// Mitsubishi GX Works2 project: DanNhanFX3G   PLC: FX3G

// global labels: Global1
VAR_GLOBAL
  SIGNAL_BOTTLE AT X000 : BOOL;
  SIGNAL_LABEL AT X001 : BOOL;
  EMERG AT X007 : BOOL;
  LABEL_PLS AT Y000 : BOOL;
  LABEL_DIR AT Y003 : BOOL;
  PushManLabel_F AT M200 : BOOL;
  PushManLabel_R AT M201 : BOOL;
  ModeAuto AT M206 : BOOL;
  Alarm AT M207 : BOOL;
  Operation AT M208 : BOOL;
  Speed_Label AT D200 : REAL;
  Length_Label AT D202 : REAL;
  Reset AT M209 : BOOL;
  Restore AT M210 : BOOL;
  LABEL_ENB AT Y004 : BOOL;
  GIRD_PLS AT Y001 : BOOL;
  RULO_PLS AT Y002 : BOOL;
  RULO_ENB AT Y006 : BOOL;
  GIRD_ENB AT Y005 : BOOL;
  FinishPLS_Label AT M8340 : BOOL;
  PRINT_ENB AT Y007 : BOOL;
  RstCountStamp AT M211 : BOOL;
  SampleTest AT M212 : BOOL;
  Counter_Stamped AT D240 : DWORD;
  Time_Label AT D250 : DWORD;
  CommandLabel AT M300 : BOOL;
  CommandLabel1 AT M301 : BOOL;
  CommandLabel2 AT M302 : BOOL;
  Com1_Label AT M303 : BOOL;
  Length_Stamp AT D206 : REAL;
  Decr_Label AT D252 : DWORD;
  Freq_Label AT D230 : REAL;
  Range_Label AT D234 : REAL;
  Range_Stamp AT D238 : REAL;
  FullStep_Label AT D212 : REAL;
  DiffTime_Label AT D208 : DINT;
  Offset_Label AT D214 : REAL;
END_VAR

// task Task_01 (event TRUE, interval 0, priority 31): POU_01
// task InterruptX000 (event I000, interval 0, priority 31): BOTTLE
// task InterruptX001 (event I100, interval 0, priority 31): LABEL
// task TimerInterrupt (event I610, interval 0, priority 31): DelayStamp

PROGRAM POU_01
VAR
  Servo1_Label : Servo;
  Servo2_Label : Servo;
  Restore_Q : BOOL;
  Timer1_Label : TON_10;
  Timer2_Label : TON_10;
  Timer_Restore : TON_10;
  TimerENB_Label : TON_10;
  TimerENB_Q : BOOL;
  TimerPrint : TON_10;
  TimerPrint_Q : BOOL;
  Pulses_Label : REAL;
  Pulses_Stamp : REAL;
  Freq_Stamp : REAL;
END_VAR
EI( TRUE );
(* Khai bao vong quay va quang duong *)
DINCP ( SIGNAL_LABEL , Counter_Stamped);
SET( SIGNAL_LABEL AND SIGNAL_BOTTLE, Alarm);
TimerPrint( IN := PRINT_ENB, PT := T#100ms, Q := TimerPrint_Q);
RST( LDP( TRUE, TimerPrint_Q), PRINT_ENB);

DEMUL( TRUE, Length_Stamp, FullStep_Label, Range_Stamp);
DEMUL( TRUE, Length_Label+Offset_Label, FullStep_Label, Range_Label);
DEMUL( TRUE, Speed_Label, FullStep_Label, Freq_Label);

DEDIV(TRUE, Range_Stamp, 160.0, Pulses_Stamp);
DEDIV(TRUE, Range_Label, 160.0, Pulses_Label);
DEDIV(TRUE, Freq_Label, 60.0, Freq_Stamp);


(* Initialize high speed counter *)
OUT_C_32( TRUE, CC238, K2147483647);
DHSCR( CommandLabel2 , REAL_TO_DINT( Pulses_Label), CN238, CommandLabel1);
(*
DSUBP( NOT FinishPLS_Label, Range_Label, C238, Pulses_Ofset);
Pulses_Label := Range_Stamp + Pulses_Ofset;*)
DPLSR(ModeAuto AND CommandLabel1, REAL_TO_DINT( Freq_Stamp), REAL_TO_DINT( Pulses_Stamp), DiffTime_Label, LABEL_PLS);
RST( LDF( TRUE, FinishPLS_Label), CommandLabel1);
(*
DPLSY( NOT ModeAuto AND (PushManLabel_F OR PushManLabel_R), 6400, Range_Stamp, LABEL_PLS);
LABEL_DIR := PushManLabel_R;
*)
Timer_Restore( IN := Restore, PT := T#5s, Q := Restore_Q );
IF Restore_Q THEN
	Speed_Label := 140.0;
	Length_Stamp := 86.0;
	Length_Label := 66.0;
	Time_Label := 300;
	Offset_Label := 2.0;
	DiffTime_Label := 20;
	FullStep_Label := 6400.0;
END_IF;

IF RstCountStamp THEN
	Counter_Stamped := 0;
END_IF;

IF Reset THEN
	Alarm := FALSE;
	Com1_Label := FALSE;
	CommandLabel1 := FALSE;
	CommandLabel2 := FALSE;
END_IF;


(*NGUYEN LY: 
Buoc 1: khi phat hien co chai, goi timer doi  ms -> run 
Buoc 2: khi het thoi gian tre -> chay Step dan het nhan.
Ly do: de danh Command1 doi chai tiep theo
Do duong kinh ong bang encoder: khi ong di qua cam bien lay xung canh len - dem encoder counter,
khi ong qua het lay xung canh xuong doc encoder counter
*)
END_PROGRAM

FUNCTION_BLOCK Servo
VAR_INPUT
  SetAutoMan : BOOL;
  Speed : DINT;
  Range : DINT;
END_VAR
VAR_IN_OUT
  SetAutoRunF : BOOL;
  SetAutoRunR : BOOL;
END_VAR
VAR_OUTPUT
  OutputPLS : BOOL;
  OutputDIR : BOOL;
END_VAR
VAR
  RelayPLS : BOOL;
  RelayDIR : BOOL;
END_VAR
VAR_IN_OUT
  PushManF : BOOL;
  PushManR : BOOL;
END_VAR
VAR_INPUT
  LimitOutput : BOOL;
  LimitInput : BOOL;
END_VAR
(* Set mode Auto/Man *)
IF  SetAutoMan THEN
	RelayDIR := SetAutoRunR;
	RelayPLS := SetAutoRunF OR SetAutoRunR;
ELSE
	RelayDIR := PushManR;
	RelayPLS := PushManF OR PushManR;
END_IF;

OutputDIR := RelayDIR ;

DPLSY( RelayPLS AND LimitInput, Speed, Range , OutputPLS );

(* Reset control signal *)
RST( LDF( TRUE, LimitOutput ) , SetAutoRunF );
RST( LDF( TRUE, LimitOutput) , SetAutoRunR );
RST( LDF( TRUE, LimitOutput ) , PushManF );
RST( LDF( TRUE, LimitOutput) , PushManR );
END_FUNCTION_BLOCK

PROGRAM BOTTLE
VAR
  Buffer : DINT;
END_VAR
DDIV( TRUE , Time_Label , 10, D500 );
DMOV(TRUE, D500, Decr_Label);
SET( TRUE, CommandLabel);
RST( TRUE, CommandLabel2);
END_PROGRAM

PROGRAM LABEL
DMOV( TRUE, 0, C238); 
SET( TRUE, CommandLabel2);
SET( TRUE, PRINT_ENB);
END_PROGRAM

PROGRAM DelayStamp
DDEC( CommandLabel, Decr_Label);
IF ModeAuto THEN
	SET( LDP( TRUE, Decr_Label <= 0), CommandLabel1);
	RST( LDP( TRUE, Decr_Label <= 0), CommandLabel); 
END_IF;
END_PROGRAM
